{attribute 'GeneratedUsingTerminal: EL3483-0060-0018'}
{attribute addProperty BoxType "EL3483-0060-0018"}
{attribute addProperty Id "VoltageAT %I*REAL4"}
{attribute addProperty CRC "2671734600"}
{attribute addProperty Size "4"}
TYPE L1_Basic_9F3F6F48 :
STRUCT
	{attribute addProperty Name "Voltage"}
	Voltage AT %I* : REAL;
END_STRUCT
END_TYPE

(* stored: Version 1.2.0.0, ProductVersion 3.1.4024.9
   DUT L1_Basic_9F3F6F48: Id {92ce4a54-74f1-498b-bea6-2455c4a3cdda} *)
